TYPE LAxisCtrl_typePosSuperimposed :
STRUCT

	distance		: LREAL;
	velocityDiff		: LREAL;
	acceleration	: LREAL;
	deceleration	: LREAL;
	jerk			: LREAL;
	direction		: DINT;

END_STRUCT
END_TYPE

(* stored: Version 1.1.0.1
   DUT LAxisCtrl_typePosSuperimposed: Id {41d110e3-e84c-4e1e-adfa-c90d4dbaa945} *)
